FUNCTION_BLOCK FB_UM_Machine EXTENDS FB_PackML_BaseModule
VAR
	// Submodules
	
	// Components
	TempController: FB_TempController	:= (Name := 'Temperature Controller');
	
	// Module Data
	// --Param
	// --Recipe
	// --HMI
	HMI: ST_HMI_Machine;
	
	// Alarms
	
	// Other I/O

	// Machine Control
	rtrigControl: R_TRIG;
	CheckAbort: BOOL;
	CheckStop: BOOL;
	
	// Miscellaneous
	
END_VAR

METHOD PROTECTED Aborted
VAR_INPUT
END_VAR
END_METHOD

METHOD PROTECTED Aborting
VAR_INPUT
END_VAR
CASE _CurrentMode OF
	E_PMLUnitMode.ePMLUnitMode_Production:
        CASE DescendantSequenceState OF
			0:
				NoStateTasksToComplete := FALSE;
				DescendantSequenceState := DescendantSequenceState + 10;
			10:
				StateTasksComplete := TRUE;
		END_CASE
		
	E_PMLUnitMode.ePMLUnitMode_Manual, E_PMLUnitMode.ePMLUnitMode_Maintenance:
        ;	
END_CASE

// Call Super
SUPER^.Aborting();
END_METHOD

METHOD PROTECTED Clearing
VAR_INPUT
END_VAR
CASE _CurrentMode OF
	E_PMLUnitMode.ePMLUnitMode_Production:
        CASE DescendantSequenceState OF
			0:
				NoStateTasksToComplete := FALSE;
				DescendantSequenceState := DescendantSequenceState + 10;
			10:
				StateTasksComplete := TRUE;
		END_CASE
		
	E_PMLUnitMode.ePMLUnitMode_Manual, E_PMLUnitMode.ePMLUnitMode_Maintenance:
        ;	
END_CASE

// Call Super
SUPER^.Clearing();
END_METHOD

METHOD PROTECTED Complete
VAR_INPUT
END_VAR
END_METHOD

//! @summary Initializes event function blocks using this module's name
METHOD PROTECTED CreateEvents

//! @description This method is called by <c>Initialize()</c> as required
// Add your event creation here

// Super call to base
SUPER^.CreateEvents();
END_METHOD

METHOD CyclicLogic
VAR_INPUT
END_VAR
IF NOT _InitComplete THEN
    _InitComplete := Initialize();
    RETURN;
END_IF

MachineControl();

SUPER^.CyclicLogic();
END_METHOD

METHOD PROTECTED Execute
VAR_INPUT
END_VAR
CASE _CurrentMode OF
	E_PMLUnitMode.ePMLUnitMode_Production:
        CASE DescendantSequenceState OF
			0:
				DescendantSequenceState := DescendantSequenceState + 10;
			10:
				;
		END_CASE
		
	E_PMLUnitMode.ePMLUnitMode_Manual, E_PMLUnitMode.ePMLUnitMode_Maintenance:
        ;	
END_CASE
END_METHOD

METHOD PROTECTED Held
VAR_INPUT
END_VAR
END_METHOD

METHOD PROTECTED Holding
VAR_INPUT
END_VAR
CASE _CurrentMode OF
	E_PMLUnitMode.ePMLUnitMode_Production:
        CASE DescendantSequenceState OF
			0:
				NoStateTasksToComplete := FALSE;
				DescendantSequenceState := DescendantSequenceState + 10;
			10:
				StateTasksComplete := TRUE;
		END_CASE
		
	E_PMLUnitMode.ePMLUnitMode_Manual, E_PMLUnitMode.ePMLUnitMode_Maintenance:
        ;	
END_CASE

// Call Super
SUPER^.Holding();
END_METHOD

METHOD PROTECTED Idle
VAR_INPUT
END_VAR
END_METHOD

//! @summary Basic module initialization logic
METHOD PROTECTED Initialize : BOOL;
VAR
	i						 : UDINT;
	varInfo					 : __SYSTEM.VAR_INFO;
	AllSubUnitsInitialized	 : BOOL := TRUE;
	AllComponentsInitialized : BOOL := TRUE;
END_VAR

//! @description This method is called by <c>CyclicLogic()</c> as required
Initialize := FALSE;
CASE DescendantSequenceState OF
    0: // Initialize
        _LogModeChanges         := FALSE;
        _LogStateChanges        := FALSE;
        DescendantSequenceState := DescendantSequenceState + 10;
	
	10: // Register Submodules
		DescendantSequenceState := DescendantSequenceState + 10;
		
    20: // Register Components
		RegisterComponent(TempController);
        DescendantSequenceState := DescendantSequenceState + 10;
		
    30: // Call the Super
        IF SUPER^.Initialize() THEN
            DescendantSequenceState := DescendantSequenceState + 10;
        END_IF
    40:
        Initialize := TRUE;
END_CASE
END_METHOD

METHOD MachineControl
VAR_INPUT
END_VAR
// Control Triggers
rtrigControl(CLK:= HMI.Command.Start XOR HMI.Command.Stop XOR HMI.Command.Reset XOR HMI.Command.Abort);

CASE CurrentState OF
	E_PMLState.ePMLState_Aborting:
		CheckAbort := FALSE;
		CheckStop := FALSE;
		
	E_PMLState.ePMLState_Aborted:
		// Wait for Reset to Clear
		IF rtrigControl.Q AND HMI.Command.Reset THEN
			ChangeState(E_PMLCommand.ePMLCommand_Clear);
		END_IF
		
	E_PMLState.ePMLState_Clearing:
		CheckAbort := TRUE;
		CheckStop := FALSE;
		
	E_PMLState.ePMLState_Stopping:
		CheckAbort := TRUE;
		CheckStop := FALSE;
		
	E_PMLState.ePMLState_Stopped:
		// Wait for Reset
		IF rtrigControl.Q AND HMI.Command.Reset THEN
			ChangeState(E_PMLCommand.ePMLCommand_Reset);
		END_IF
		
	E_PMLState.ePMLState_Resetting:
		CheckAbort := TRUE;
		CheckStop := TRUE;
	
	E_PMLState.ePMLState_Idle:
		// Wait for Start
		IF rtrigControl.Q AND HMI.Command.Start THEN
			ChangeState(E_PMLCommand.ePMLCommand_Start);
		END_IF
	
END_CASE

// Check for Abort or Stop
IF rtrigControl.Q AND HMI.Command.Abort THEN
	ChangeState(E_PMLCommand.ePMLCommand_Abort);
ELSIF rtrigControl.Q AND HMI.Command.Stop THEN
	ChangeState(E_PMLCommand.ePMLCommand_Stop);
END_IF
END_METHOD

METHOD PROTECTED Resetting
VAR_INPUT
END_VAR
CASE _CurrentMode OF
	E_PMLUnitMode.ePMLUnitMode_Production:
        CASE DescendantSequenceState OF
			0:
				NoStateTasksToComplete := FALSE;
				DescendantSequenceState := DescendantSequenceState + 10;
			10:
				StateTasksComplete := TRUE;
		END_CASE
		
	E_PMLUnitMode.ePMLUnitMode_Manual, E_PMLUnitMode.ePMLUnitMode_Maintenance:
        ;	
END_CASE

// Call Super
SUPER^.Resetting();
END_METHOD

METHOD PROTECTED Starting
VAR_INPUT
END_VAR
CASE _CurrentMode OF
	E_PMLUnitMode.ePMLUnitMode_Production:
        CASE DescendantSequenceState OF
			0:
				NoStateTasksToComplete := FALSE;
				DescendantSequenceState := DescendantSequenceState + 10;
			10:
				StateTasksComplete := TRUE;
		END_CASE
		
	E_PMLUnitMode.ePMLUnitMode_Manual, E_PMLUnitMode.ePMLUnitMode_Maintenance:
        ;	
END_CASE

// Call Super
SUPER^.Starting();
END_METHOD

METHOD PROTECTED Stopped
VAR_INPUT
END_VAR
END_METHOD

METHOD PROTECTED Stopping
VAR_INPUT
END_VAR
CASE _CurrentMode OF
	E_PMLUnitMode.ePMLUnitMode_Production:
        CASE DescendantSequenceState OF
			0:
				NoStateTasksToComplete := FALSE;
				DescendantSequenceState := DescendantSequenceState + 10;
			10:
				StateTasksComplete := TRUE;
		END_CASE
		
	E_PMLUnitMode.ePMLUnitMode_Manual, E_PMLUnitMode.ePMLUnitMode_Maintenance:
        ;	
END_CASE

// Call Super
SUPER^.Stopping();
END_METHOD

METHOD PROTECTED Suspended
VAR_INPUT
END_VAR
END_METHOD

METHOD PROTECTED Suspending
VAR_INPUT
END_VAR
CASE _CurrentMode OF
	E_PMLUnitMode.ePMLUnitMode_Production:
        CASE DescendantSequenceState OF
			0:
				NoStateTasksToComplete := FALSE;
				DescendantSequenceState := DescendantSequenceState + 10;
			10:
				StateTasksComplete := TRUE;
		END_CASE
		
	E_PMLUnitMode.ePMLUnitMode_Manual, E_PMLUnitMode.ePMLUnitMode_Maintenance:
        ;	
END_CASE

// Call Super
SUPER^.Suspending();
END_METHOD

METHOD PROTECTED Undefined
VAR_INPUT
END_VAR
END_METHOD

METHOD PROTECTED Unholding
VAR_INPUT
END_VAR
CASE _CurrentMode OF
	E_PMLUnitMode.ePMLUnitMode_Production:
        CASE DescendantSequenceState OF
			0:
				NoStateTasksToComplete := FALSE;
				DescendantSequenceState := DescendantSequenceState + 10;
			10:
				StateTasksComplete := TRUE;
		END_CASE
		
	E_PMLUnitMode.ePMLUnitMode_Manual, E_PMLUnitMode.ePMLUnitMode_Maintenance:
        ;	
END_CASE

// Call Super
SUPER^.Unholding();
END_METHOD

METHOD PROTECTED Unsuspending
VAR_INPUT
END_VAR
CASE _CurrentMode OF
	E_PMLUnitMode.ePMLUnitMode_Production:
        CASE DescendantSequenceState OF
			0:
				NoStateTasksToComplete := FALSE;
				DescendantSequenceState := DescendantSequenceState + 10;
			10:
				StateTasksComplete := TRUE;
		END_CASE
		
	E_PMLUnitMode.ePMLUnitMode_Manual, E_PMLUnitMode.ePMLUnitMode_Maintenance:
        ;	
END_CASE

// Call Super
SUPER^.Unsuspending();
END_METHOD

END_FUNCTION_BLOCK

(* stored: Version 1.1.0.1, ProductVersion 3.1.4024.12
   POU FB_UM_Machine: Id {92d579da-ce14-4975-99e5-d28fcc6e3c29}, SpecialFunc None
   Folder PackML: Id {eba94962-0d0a-46b4-bc0a-8b3c13da286f}
   Folder Acting States: Id {0611eaea-d8fa-404c-9043-aa64112d6399}
   Folder Waiting States: Id {2faa95d5-bfa2-474f-bef7-b1e460095506}
   Folder REFs: Id {457947ab-d7f0-4d25-818d-d5fe85adf09e}
   Method Aborted: Id {0f799341-08d3-4eb7-ba2d-8c71ba0c6431}
   Method Aborting: Id {98dcd633-3854-4540-b758-997508b7c91b}
   Method Clearing: Id {c414fe1f-3dd8-49f8-896f-621ce691e2fa}
   Method Complete: Id {ec8c24e1-5604-4f4b-8e9a-19cd915062ff}
   Method CreateEvents: Id {16295d0b-7aa6-4f8a-b9c3-d84cdc8fcccc}
   Method CyclicLogic: Id {89674960-c11e-45f8-9e82-56fc2851f90e}
   Method Execute: Id {1083b932-ed78-476c-b3e9-6fad683f695e}
   Method Held: Id {d52971ff-c8d7-4de5-9ec9-701666d09180}
   Method Holding: Id {3cae1643-f617-4cf9-8c8e-2ff5e5cd2e84}
   Method Idle: Id {c327d264-0e29-450f-ae5b-a550621a88ee}
   Method Initialize: Id {fb842b60-6973-4924-ae95-1515cf575652}
   Method MachineControl: Id {993524d3-519c-4b5d-8509-f46920421f32}
   Method Resetting: Id {1d3174a9-ac96-459d-9a9f-2240da648282}
   Method Starting: Id {7c8d9ca9-b896-496a-b87c-5dae3e7cfde1}
   Method Stopped: Id {dcf1e622-af75-46a3-a24e-31ec5fdb9336}
   Method Stopping: Id {c3fdafe5-36d0-498d-b9fc-e2839e70822c}
   Method Suspended: Id {eecd553c-c328-4a0e-972d-87120c60cdde}
   Method Suspending: Id {94bffd1b-b501-4e6c-9da7-704d67323c69}
   Method Undefined: Id {0767a7fb-d065-4780-917b-11f3d40faf88}
   Method Unholding: Id {6dfce679-cd50-40ed-ae49-9efa2bb74fe4}
   Method Unsuspending: Id {cd191a94-977d-465e-8b83-0fe4cd0cbab9} *)
